FUNCTION_BLOCK AxesIOWidget
VAR_INPUT
END_VAR
VAR_OUTPUT
END_VAR
VAR
	actualStatus : StatusWidget;
END_VAR
VAR_IN_OUT
	ref : AxesIO;
END_VAR

actualStatus(text  := ref.actualStatus,
             color := HealthToColor(ref.statuses.healthStatus));

END_FUNCTION_BLOCK

(* stored: Version 1.1.0.1, ProductVersion 3.1.4018.5
   POU AxesIOWidget: Id {022afcb2-7b1e-47fe-bc2a-502f68050d73}, SpecialFunc None *)
